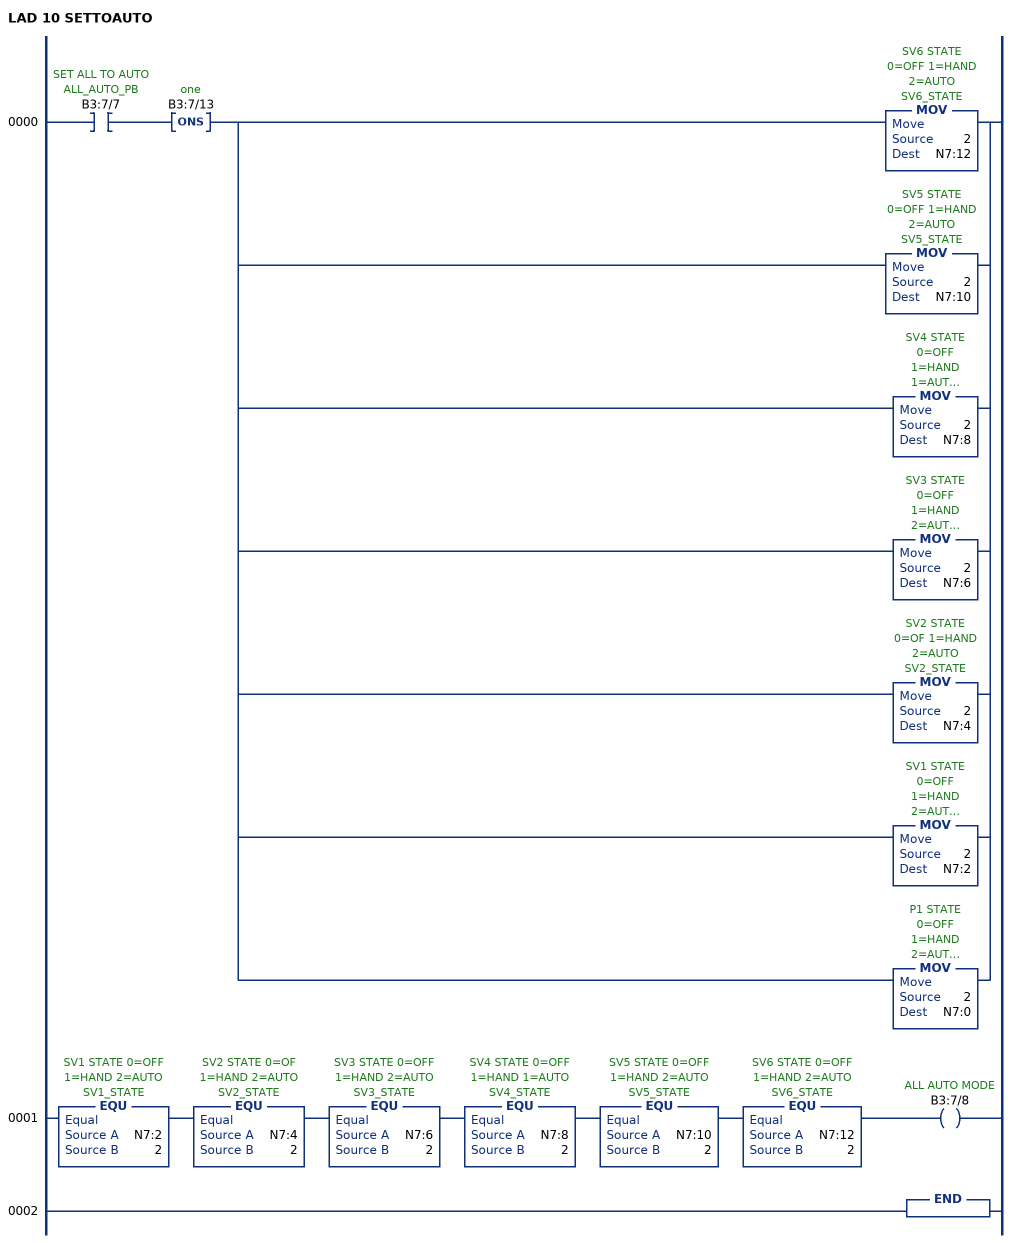
% Rung: 0 %
SOR XIC B3:7/7 ONS B3:7/13 BST MOV 2 N7:12 NXB MOV 2 N7:10 NXB MOV 2 N7:8 NXB MOV 2 N7:6 NXB MOV 2 N7:4 NXB MOV 2 N7:2 NXB MOV 2 N7:0 BND EOR
%   B3:7/7  ALL_AUTO_PB  "SET ALL TO AUTO" %
%   B3:7/13  "one" %
%   N7:12  SV6_STATE  "SV6 STATE 0=OFF 1=HAND 2=AUTO" %
%   N7:10  SV5_STATE  "SV5 STATE 0=OFF 1=HAND 2=AUTO" %
%   N7:8  SV4_STATE  "SV4 STATE 0=OFF 1=HAND 1=AUTO" %
%   N7:6  SV3_STATE  "SV3 STATE 0=OFF 1=HAND 2=AUTO" %
%   N7:4  SV2_STATE  "SV2 STATE 0=OF 1=HAND 2=AUTO" %
%   N7:2  SV1_STATE  "SV1 STATE 0=OFF 1=HAND 2=AUTO" %
%   N7:0  P1_STATE  "P1 STATE 0=OFF 1=HAND 2=AUTO" %
% Rung: 1 %
SOR EQU N7:2 2 EQU N7:4 2 EQU N7:6 2 EQU N7:8 2 EQU N7:10 2 EQU N7:12 2 OTE B3:7/8 EOR
%   N7:2  SV1_STATE  "SV1 STATE 0=OFF 1=HAND 2=AUTO" %
%   N7:4  SV2_STATE  "SV2 STATE 0=OF 1=HAND 2=AUTO" %
%   N7:6  SV3_STATE  "SV3 STATE 0=OFF 1=HAND 2=AUTO" %
%   N7:8  SV4_STATE  "SV4 STATE 0=OFF 1=HAND 1=AUTO" %
%   N7:10  SV5_STATE  "SV5 STATE 0=OFF 1=HAND 2=AUTO" %
%   N7:12  SV6_STATE  "SV6 STATE 0=OFF 1=HAND 2=AUTO" %
%   B3:7/8  "ALL AUTO MODE" %
% Rung: 2 %
SOR END EOR

OTHER DOCUMENTED ADDRESSES
  B3:4/11  "PUMP ON"
  I:0.0/0  "SV1 ip"
  I:0.0/1  "SV1 ip"
  I:0.0/2  "SV2 ip"
  I:0.0/3  "SV3 ip"
  I:0.0/4  "SV4 ip"
  I:0.0/5  "SV5 ip"
  I:0.0/6  "SV6 ip"
  I:1.0/0  "Pressure transmitter PT1 (psi)"
  T4:2.ACC  SECONDS

DATA TABLE (non-zero values as saved)
DATA T4
% .PRE .ACC %
% T4:0 % 10 0
% T4:1 % 10 0
% T4:2 % 60 0
% T4:3 % 10 0
% T4:4 % 60 0
% T4:5 % 5 0
% T4:6 % 5 0
% T4:7 % 10 0
% T4:8 % 10 0
% T4:9 % 10 0
% T4:10 % 3 0
DATA F8
% F8:0 % 0.5 0.5 0 0 0
% F8:5 % 0 12 90 15 15
